FUNCTION_BLOCK PUBLISH_0 (* Event-only Publisher *)
  (* Standard: 61499-2 *)
  (* Version 0.2, 2001-01-27, JHC, Rockwell Automation, Added no_double_init, reinitialize. *)
  (* Version 0.1, 2000-03-23, JHC, Rockwell Automation, NULL encoding fixed. *)
  (* Compiler header: package fb.rt.net; *)
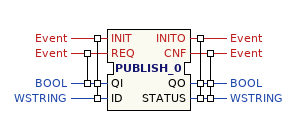
  EVENT_INPUT
    INIT WITH QI, ID; (* Service Initialization *)
    REQ WITH QI; (* Service Request *)
  END_EVENT
  EVENT_OUTPUT
    INITO WITH QO, STATUS; (* Initialization Confirm *)
    CNF WITH QO, STATUS; (* Service Confirmation *)
  END_EVENT
  VAR_INPUT
    QI : BOOL; (* Event Input Qualifier *)
    ID : WSTRING; (* Connection Identifier *)
  END_VAR
  VAR_OUTPUT
    QO : BOOL; (* Event Output Qualifier *)
    STATUS : WSTRING; (* Service Status *)
  END_VAR
  SERVICE PUBLISH_0/SUBSCRIBE_0 (* Event Publication Service *)
    SEQUENCE normal_establishment
      PUBLISH_0.INIT+(ID) -> PUBLISH_0.INITO+();
      SUBSCRIBE_0.INIT+(ID) -> SUBSCRIBE_0.INITO+();
    END_SEQUENCE
    SEQUENCE no_double_init
      PUBLISH_0.INIT+(ID) -> PUBLISH_0.INITO+(STATUS);
      PUBLISH_0.INIT+(ID);
    END_SEQUENCE
    SEQUENCE reinitialize
      PUBLISH_0.INIT+(ID) -> PUBLISH_0.INITO+();
      PUBLISH_0.INIT-() -> PUBLISH_0.INITO-(STATUS);
      PUBLISH_0.INIT+(ID) -> PUBLISH_0.INITO+();
    END_SEQUENCE
    SEQUENCE publisher_rejected_establishment
      PUBLISH_0.INIT+(ID) -> PUBLISH_0.INITO-(STATUS);
    END_SEQUENCE
    SEQUENCE subscriber_rejected_establishment
      SUBSCRIBE_0.INIT+(ID) -> SUBSCRIBE_0.INITO-(STATUS);
    END_SEQUENCE
    SEQUENCE event_transfer
      PUBLISH_0.REQ+() -> SUBSCRIBE_0.IND+();
      -> PUBLISH_0.CNF+();
      SUBSCRIBE_0.RSP+();
    END_SEQUENCE
    SEQUENCE publisher_initiated_disconnect
      PUBLISH_0.INIT-() -> SUBSCRIBE_0.INITO-(STATUS);
      -> PUBLISH_0.INITO-(STATUS);
    END_SEQUENCE
    SEQUENCE subscriber_initiated_disconnect
      SUBSCRIBE_0.INIT-() -> SUBSCRIBE_0.INITO-(STATUS);
    END_SEQUENCE
    SEQUENCE system_publisher_disconnect
      -> PUBLISH_0.INITO-(STATUS);
      -> SUBSCRIBE_0.INITO-(STATUS);
    END_SEQUENCE
    SEQUENCE system_subscriber_disconnect
      -> SUBSCRIBE_0.INITO-(STATUS);
    END_SEQUENCE
  END_SERVICE
END_FUNCTION_BLOCK
